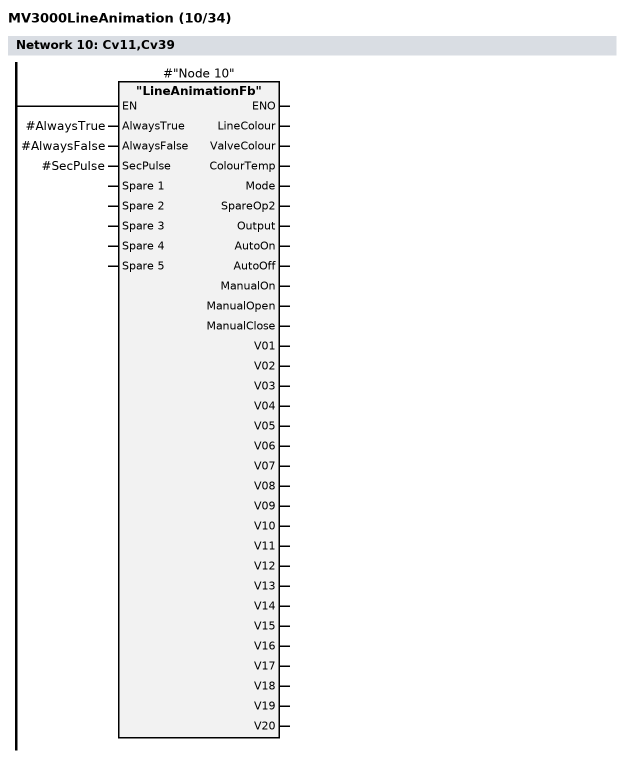
   RUNG wire#powerrail
      #"Node 10"(AlwaysTrue := #AlwaysTrue, AlwaysFalse := #AlwaysFalse, SecPulse := #SecPulse, "Spare 1" :=, "Spare 2" :=, "Spare 3" :=, "Spare 4" :=, "Spare 5" :=, LineColour =>, ValveColour =>, ColourTemp =>, Mode =>, SpareOp2 =>, Output =>, AutoOn =>, AutoOff =>, ManualOn =>, ManualOpen =>, ManualClose =>, V01 =>, V02 =>, V03 =>, V04 =>, V05 =>, V06 =>, V07 =>, V08 =>, V09 =>, V10 =>, V11 =>, V12 =>, V13 =>, V14 =>, V15 =>, V16 =>, V17 =>, V18 =>, V19 =>, V20 =>)
   END_RUNG
   // the same network as SCL:
   #"Node 10"(AlwaysTrue := #AlwaysTrue, AlwaysFalse := #AlwaysFalse, SecPulse := #SecPulse);   // "LineAnimationFb"
END_REGION

REGION Network 11: Cv12,Cv64, Cv26
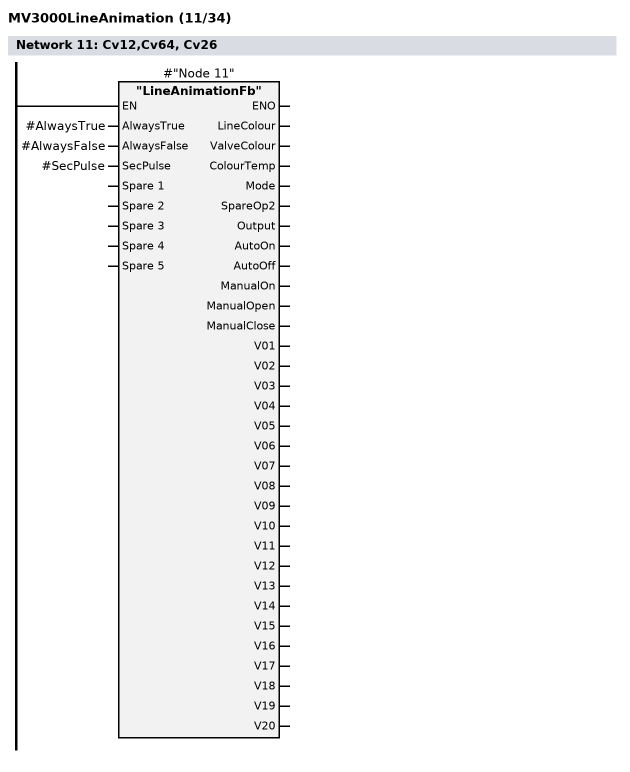
   RUNG wire#powerrail
      #"Node 11"(AlwaysTrue := #AlwaysTrue, AlwaysFalse := #AlwaysFalse, SecPulse := #SecPulse, "Spare 1" :=, "Spare 2" :=, "Spare 3" :=, "Spare 4" :=, "Spare 5" :=, LineColour =>, ValveColour =>, ColourTemp =>, Mode =>, SpareOp2 =>, Output =>, AutoOn =>, AutoOff =>, ManualOn =>, ManualOpen =>, ManualClose =>, V01 =>, V02 =>, V03 =>, V04 =>, V05 =>, V06 =>, V07 =>, V08 =>, V09 =>, V10 =>, V11 =>, V12 =>, V13 =>, V14 =>, V15 =>, V16 =>, V17 =>, V18 =>, V19 =>, V20 =>)
   END_RUNG
   // the same network as SCL:
   #"Node 11"(AlwaysTrue := #AlwaysTrue, AlwaysFalse := #AlwaysFalse, SecPulse := #SecPulse);   // "LineAnimationFb"
END_REGION

REGION Network 12: Cv31,Cv41
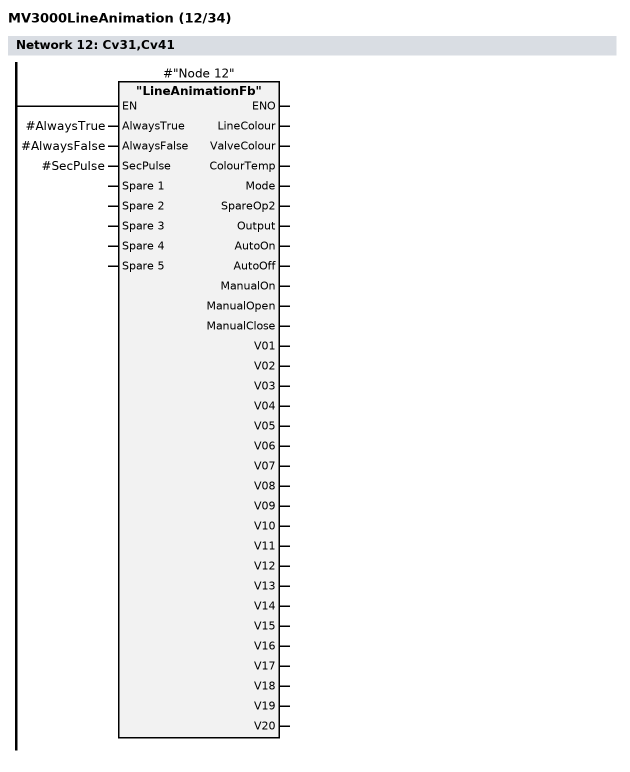
   RUNG wire#powerrail
      #"Node 12"(AlwaysTrue := #AlwaysTrue, AlwaysFalse := #AlwaysFalse, SecPulse := #SecPulse, "Spare 1" :=, "Spare 2" :=, "Spare 3" :=, "Spare 4" :=, "Spare 5" :=, LineColour =>, ValveColour =>, ColourTemp =>, Mode =>, SpareOp2 =>, Output =>, AutoOn =>, AutoOff =>, ManualOn =>, ManualOpen =>, ManualClose =>, V01 =>, V02 =>, V03 =>, V04 =>, V05 =>, V06 =>, V07 =>, V08 =>, V09 =>, V10 =>, V11 =>, V12 =>, V13 =>, V14 =>, V15 =>, V16 =>, V17 =>, V18 =>, V19 =>, V20 =>)
   END_RUNG
   // the same network as SCL:
   #"Node 12"(AlwaysTrue := #AlwaysTrue, AlwaysFalse := #AlwaysFalse, SecPulse := #SecPulse);   // "LineAnimationFb"
END_REGION

REGION Network 13: Fbov01, cV30 ,CV31 , CV 32 , CV33
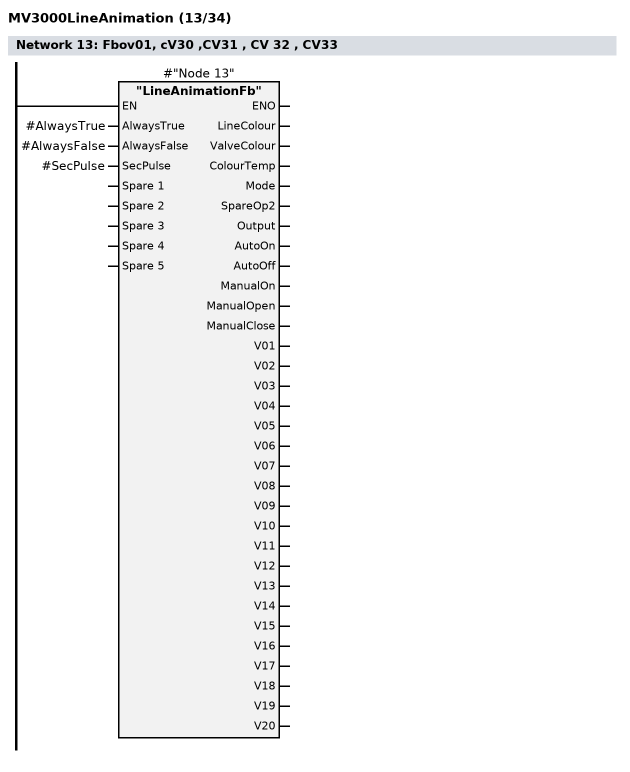
   RUNG wire#powerrail
      #"Node 13"(AlwaysTrue := #AlwaysTrue, AlwaysFalse := #AlwaysFalse, SecPulse := #SecPulse, "Spare 1" :=, "Spare 2" :=, "Spare 3" :=, "Spare 4" :=, "Spare 5" :=, LineColour =>, ValveColour =>, ColourTemp =>, Mode =>, SpareOp2 =>, Output =>, AutoOn =>, AutoOff =>, ManualOn =>, ManualOpen =>, ManualClose =>, V01 =>, V02 =>, V03 =>, V04 =>, V05 =>, V06 =>, V07 =>, V08 =>, V09 =>, V10 =>, V11 =>, V12 =>, V13 =>, V14 =>, V15 =>, V16 =>, V17 =>, V18 =>, V19 =>, V20 =>)
   END_RUNG
   // the same network as SCL:
   #"Node 13"(AlwaysTrue := #AlwaysTrue, AlwaysFalse := #AlwaysFalse, SecPulse := #SecPulse);   // "LineAnimationFb"
END_REGION

REGION Network 14: CV27 ,CV 28 ,CV 29
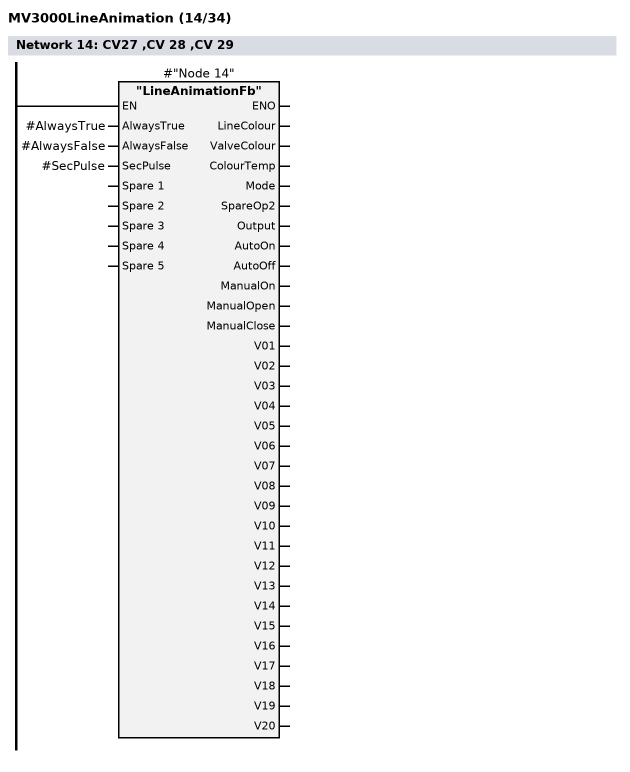
   RUNG wire#powerrail
      #"Node 14"(AlwaysTrue := #AlwaysTrue, AlwaysFalse := #AlwaysFalse, SecPulse := #SecPulse, "Spare 1" :=, "Spare 2" :=, "Spare 3" :=, "Spare 4" :=, "Spare 5" :=, LineColour =>, ValveColour =>, ColourTemp =>, Mode =>, SpareOp2 =>, Output =>, AutoOn =>, AutoOff =>, ManualOn =>, ManualOpen =>, ManualClose =>, V01 =>, V02 =>, V03 =>, V04 =>, V05 =>, V06 =>, V07 =>, V08 =>, V09 =>, V10 =>, V11 =>, V12 =>, V13 =>, V14 =>, V15 =>, V16 =>, V17 =>, V18 =>, V19 =>, V20 =>)
   END_RUNG
   // the same network as SCL:
   #"Node 14"(AlwaysTrue := #AlwaysTrue, AlwaysFalse := #AlwaysFalse, SecPulse := #SecPulse);   // "LineAnimationFb"
END_REGION

REGION Network 15: CV30 ,CV 33 ,CV 34,CV 35
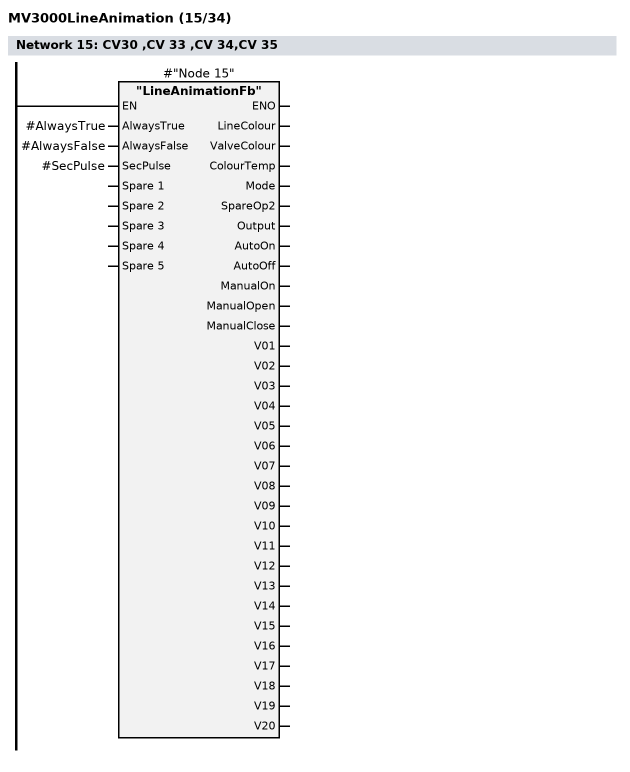
   RUNG wire#powerrail
      #"Node 15"(AlwaysTrue := #AlwaysTrue, AlwaysFalse := #AlwaysFalse, SecPulse := #SecPulse, "Spare 1" :=, "Spare 2" :=, "Spare 3" :=, "Spare 4" :=, "Spare 5" :=, LineColour =>, ValveColour =>, ColourTemp =>, Mode =>, SpareOp2 =>, Output =>, AutoOn =>, AutoOff =>, ManualOn =>, ManualOpen =>, ManualClose =>, V01 =>, V02 =>, V03 =>, V04 =>, V05 =>, V06 =>, V07 =>, V08 =>, V09 =>, V10 =>, V11 =>, V12 =>, V13 =>, V14 =>, V15 =>, V16 =>, V17 =>, V18 =>, V19 =>, V20 =>)
   END_RUNG
   // the same network as SCL:
   #"Node 15"(AlwaysTrue := #AlwaysTrue, AlwaysFalse := #AlwaysFalse, SecPulse := #SecPulse);   // "LineAnimationFb"
END_REGION

REGION Network 16: CV32 ,CV 36 ,CV 39,CV 40
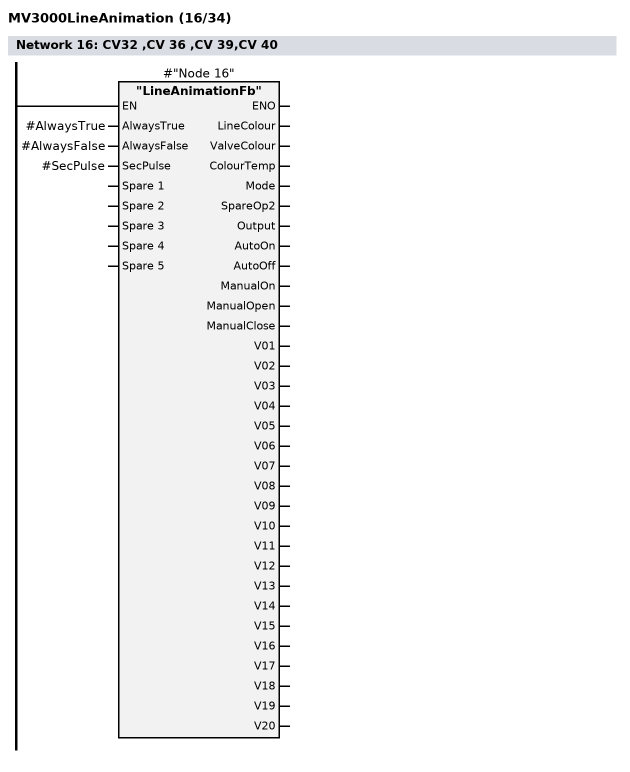
   RUNG wire#powerrail
      #"Node 16"(AlwaysTrue := #AlwaysTrue, AlwaysFalse := #AlwaysFalse, SecPulse := #SecPulse, "Spare 1" :=, "Spare 2" :=, "Spare 3" :=, "Spare 4" :=, "Spare 5" :=, LineColour =>, ValveColour =>, ColourTemp =>, Mode =>, SpareOp2 =>, Output =>, AutoOn =>, AutoOff =>, ManualOn =>, ManualOpen =>, ManualClose =>, V01 =>, V02 =>, V03 =>, V04 =>, V05 =>, V06 =>, V07 =>, V08 =>, V09 =>, V10 =>, V11 =>, V12 =>, V13 =>, V14 =>, V15 =>, V16 =>, V17 =>, V18 =>, V19 =>, V20 =>)
   END_RUNG
   // the same network as SCL:
   #"Node 16"(AlwaysTrue := #AlwaysTrue, AlwaysFalse := #AlwaysFalse, SecPulse := #SecPulse);   // "LineAnimationFb"
END_REGION

REGION Network 17: CV40 ,CV41 ,CV 42 ,CV 43,CV 44
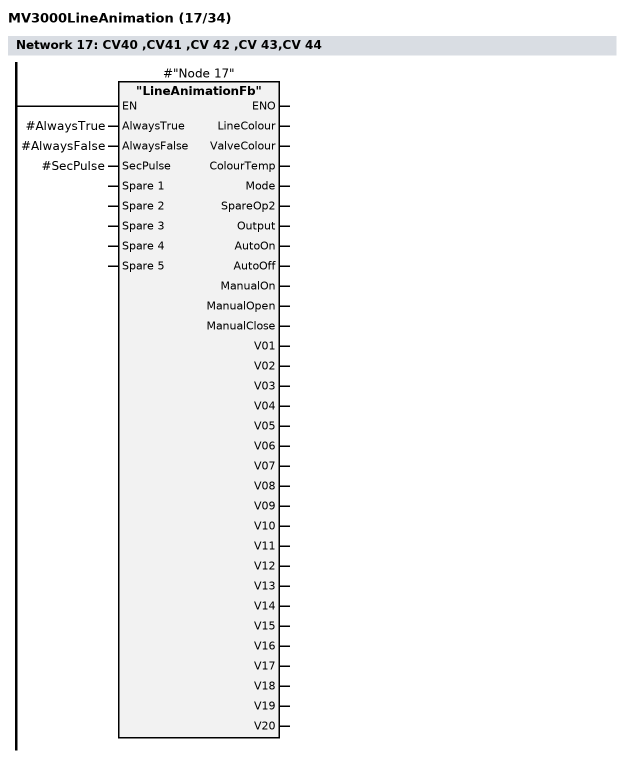
   RUNG wire#powerrail
      #"Node 17"(AlwaysTrue := #AlwaysTrue, AlwaysFalse := #AlwaysFalse, SecPulse := #SecPulse, "Spare 1" :=, "Spare 2" :=, "Spare 3" :=, "Spare 4" :=, "Spare 5" :=, LineColour =>, ValveColour =>, ColourTemp =>, Mode =>, SpareOp2 =>, Output =>, AutoOn =>, AutoOff =>, ManualOn =>, ManualOpen =>, ManualClose =>, V01 =>, V02 =>, V03 =>, V04 =>, V05 =>, V06 =>, V07 =>, V08 =>, V09 =>, V10 =>, V11 =>, V12 =>, V13 =>, V14 =>, V15 =>, V16 =>, V17 =>, V18 =>, V19 =>, V20 =>)
   END_RUNG
   // the same network as SCL:
   #"Node 17"(AlwaysTrue := #AlwaysTrue, AlwaysFalse := #AlwaysFalse, SecPulse := #SecPulse);   // "LineAnimationFb"
END_REGION

REGION Network 18: CV43 ,CV47 ,CV 48 ,CV 49,CV 50
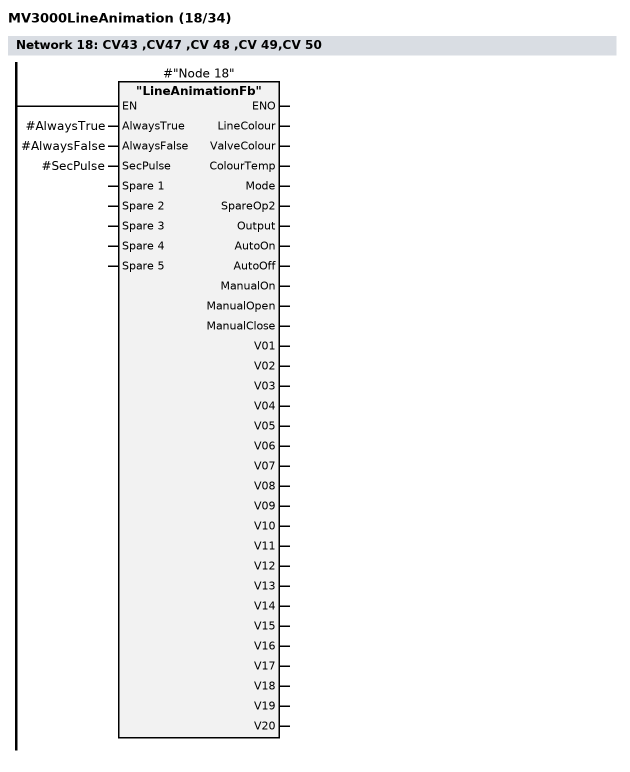
   RUNG wire#powerrail
      #"Node 18"(AlwaysTrue := #AlwaysTrue, AlwaysFalse := #AlwaysFalse, SecPulse := #SecPulse, "Spare 1" :=, "Spare 2" :=, "Spare 3" :=, "Spare 4" :=, "Spare 5" :=, LineColour =>, ValveColour =>, ColourTemp =>, Mode =>, SpareOp2 =>, Output =>, AutoOn =>, AutoOff =>, ManualOn =>, ManualOpen =>, ManualClose =>, V01 =>, V02 =>, V03 =>, V04 =>, V05 =>, V06 =>, V07 =>, V08 =>, V09 =>, V10 =>, V11 =>, V12 =>, V13 =>, V14 =>, V15 =>, V16 =>, V17 =>, V18 =>, V19 =>, V20 =>)
   END_RUNG
   // the same network as SCL:
   #"Node 18"(AlwaysTrue := #AlwaysTrue, AlwaysFalse := #AlwaysFalse, SecPulse := #SecPulse);   // "LineAnimationFb"
END_REGION

REGION Network 19: CV49 ,CV53 ,CV 54 ,CV 55,CV 56
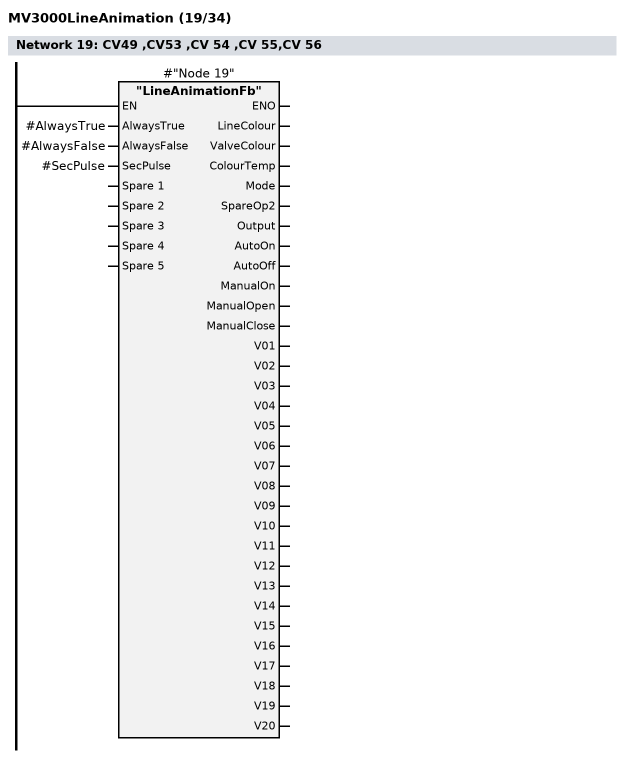
   RUNG wire#powerrail
      #"Node 19"(AlwaysTrue := #AlwaysTrue, AlwaysFalse := #AlwaysFalse, SecPulse := #SecPulse, "Spare 1" :=, "Spare 2" :=, "Spare 3" :=, "Spare 4" :=, "Spare 5" :=, LineColour =>, ValveColour =>, ColourTemp =>, Mode =>, SpareOp2 =>, Output =>, AutoOn =>, AutoOff =>, ManualOn =>, ManualOpen =>, ManualClose =>, V01 =>, V02 =>, V03 =>, V04 =>, V05 =>, V06 =>, V07 =>, V08 =>, V09 =>, V10 =>, V11 =>, V12 =>, V13 =>, V14 =>, V15 =>, V16 =>, V17 =>, V18 =>, V19 =>, V20 =>)
   END_RUNG
   // the same network as SCL:
   #"Node 19"(AlwaysTrue := #AlwaysTrue, AlwaysFalse := #AlwaysFalse, SecPulse := #SecPulse);   // "LineAnimationFb"
END_REGION

REGION Network 20: Cv55,Cv61, Cv62
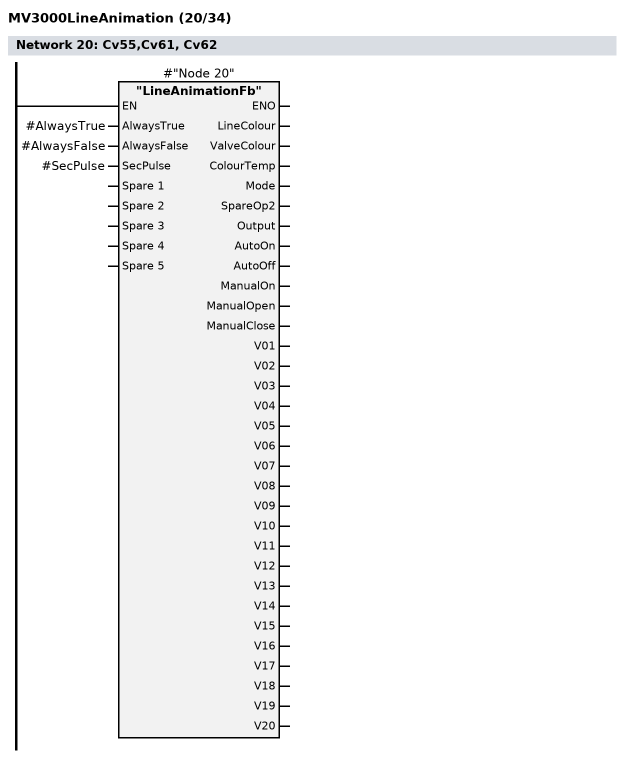
   RUNG wire#powerrail
      #"Node 20"(AlwaysTrue := #AlwaysTrue, AlwaysFalse := #AlwaysFalse, SecPulse := #SecPulse, "Spare 1" :=, "Spare 2" :=, "Spare 3" :=, "Spare 4" :=, "Spare 5" :=, LineColour =>, ValveColour =>, ColourTemp =>, Mode =>, SpareOp2 =>, Output =>, AutoOn =>, AutoOff =>, ManualOn =>, ManualOpen =>, ManualClose =>, V01 =>, V02 =>, V03 =>, V04 =>, V05 =>, V06 =>, V07 =>, V08 =>, V09 =>, V10 =>, V11 =>, V12 =>, V13 =>, V14 =>, V15 =>, V16 =>, V17 =>, V18 =>, V19 =>, V20 =>)
   END_RUNG
   // the same network as SCL:
   #"Node 20"(AlwaysTrue := #AlwaysTrue, AlwaysFalse := #AlwaysFalse, SecPulse := #SecPulse);   // "LineAnimationFb"
END_REGION

REGION Network 21: Cv59,Cv60, Cv61
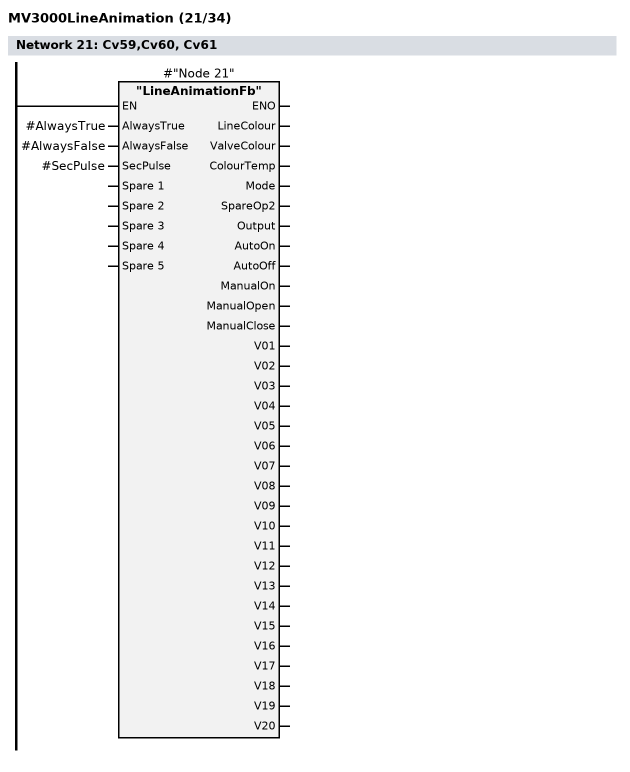
   RUNG wire#powerrail
      #"Node 21"(AlwaysTrue := #AlwaysTrue, AlwaysFalse := #AlwaysFalse, SecPulse := #SecPulse, "Spare 1" :=, "Spare 2" :=, "Spare 3" :=, "Spare 4" :=, "Spare 5" :=, LineColour =>, ValveColour =>, ColourTemp =>, Mode =>, SpareOp2 =>, Output =>, AutoOn =>, AutoOff =>, ManualOn =>, ManualOpen =>, ManualClose =>, V01 =>, V02 =>, V03 =>, V04 =>, V05 =>, V06 =>, V07 =>, V08 =>, V09 =>, V10 =>, V11 =>, V12 =>, V13 =>, V14 =>, V15 =>, V16 =>, V17 =>, V18 =>, V19 =>, V20 =>)
   END_RUNG
   // the same network as SCL:
   #"Node 21"(AlwaysTrue := #AlwaysTrue, AlwaysFalse := #AlwaysFalse, SecPulse := #SecPulse);   // "LineAnimationFb"
END_REGION

REGION Network 22: Cv56,Cv58, Cv57
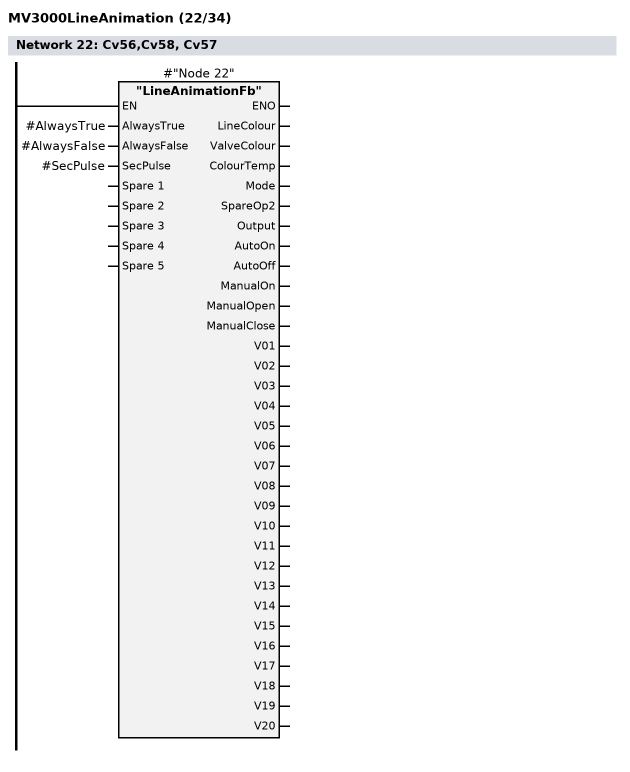
   RUNG wire#powerrail
      #"Node 22"(AlwaysTrue := #AlwaysTrue, AlwaysFalse := #AlwaysFalse, SecPulse := #SecPulse, "Spare 1" :=, "Spare 2" :=, "Spare 3" :=, "Spare 4" :=, "Spare 5" :=, LineColour =>, ValveColour =>, ColourTemp =>, Mode =>, SpareOp2 =>, Output =>, AutoOn =>, AutoOff =>, ManualOn =>, ManualOpen =>, ManualClose =>, V01 =>, V02 =>, V03 =>, V04 =>, V05 =>, V06 =>, V07 =>, V08 =>, V09 =>, V10 =>, V11 =>, V12 =>, V13 =>, V14 =>, V15 =>, V16 =>, V17 =>, V18 =>, V19 =>, V20 =>)
   END_RUNG
   // the same network as SCL:
   #"Node 22"(AlwaysTrue := #AlwaysTrue, AlwaysFalse := #AlwaysFalse, SecPulse := #SecPulse);   // "LineAnimationFb"
END_REGION

REGION Network 23: Cv50,Cv51, Cv52,Cv53
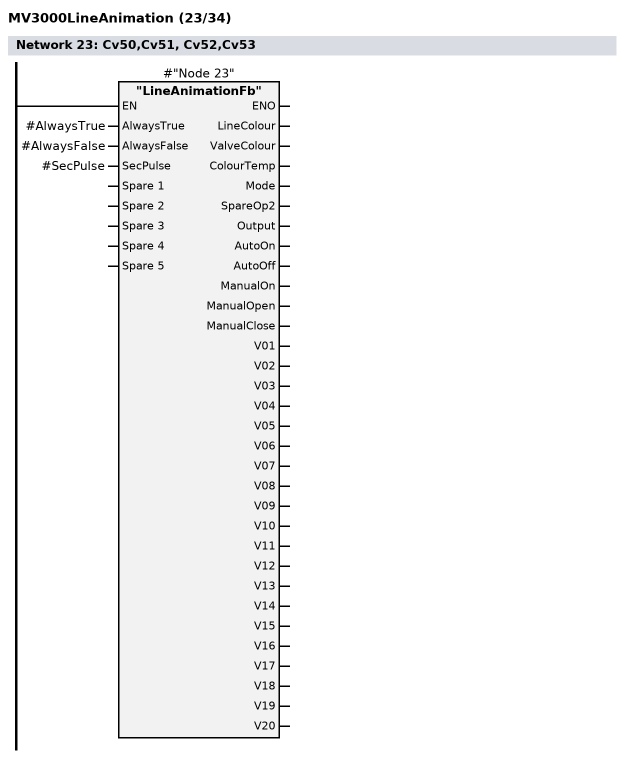
   RUNG wire#powerrail
      #"Node 23"(AlwaysTrue := #AlwaysTrue, AlwaysFalse := #AlwaysFalse, SecPulse := #SecPulse, "Spare 1" :=, "Spare 2" :=, "Spare 3" :=, "Spare 4" :=, "Spare 5" :=, LineColour =>, ValveColour =>, ColourTemp =>, Mode =>, SpareOp2 =>, Output =>, AutoOn =>, AutoOff =>, ManualOn =>, ManualOpen =>, ManualClose =>, V01 =>, V02 =>, V03 =>, V04 =>, V05 =>, V06 =>, V07 =>, V08 =>, V09 =>, V10 =>, V11 =>, V12 =>, V13 =>, V14 =>, V15 =>, V16 =>, V17 =>, V18 =>, V19 =>, V20 =>)
   END_RUNG
   // the same network as SCL:
   #"Node 23"(AlwaysTrue := #AlwaysTrue, AlwaysFalse := #AlwaysFalse, SecPulse := #SecPulse);   // "LineAnimationFb"
END_REGION

REGION Network 24: Cv44,Cv45, Cv46,Cv47
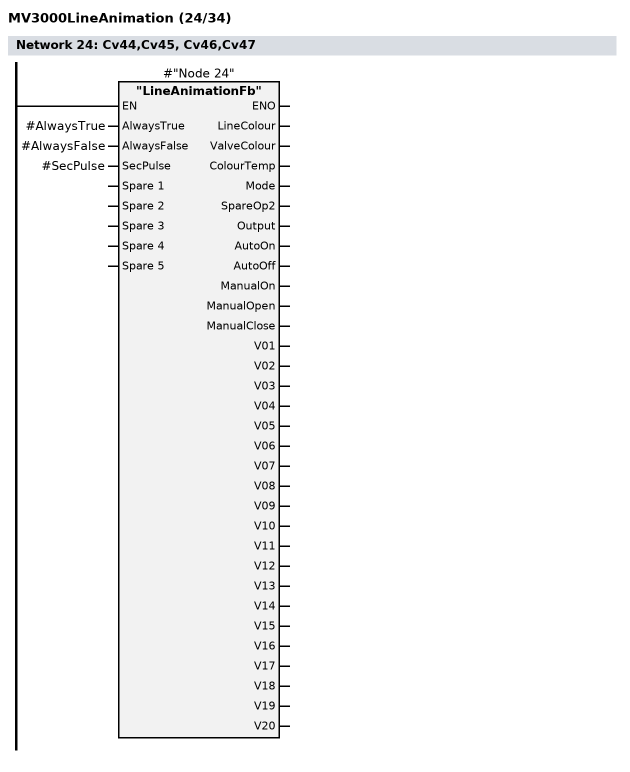
   RUNG wire#powerrail
      #"Node 24"(AlwaysTrue := #AlwaysTrue, AlwaysFalse := #AlwaysFalse, SecPulse := #SecPulse, "Spare 1" :=, "Spare 2" :=, "Spare 3" :=, "Spare 4" :=, "Spare 5" :=, LineColour =>, ValveColour =>, ColourTemp =>, Mode =>, SpareOp2 =>, Output =>, AutoOn =>, AutoOff =>, ManualOn =>, ManualOpen =>, ManualClose =>, V01 =>, V02 =>, V03 =>, V04 =>, V05 =>, V06 =>, V07 =>, V08 =>, V09 =>, V10 =>, V11 =>, V12 =>, V13 =>, V14 =>, V15 =>, V16 =>, V17 =>, V18 =>, V19 =>, V20 =>)
   END_RUNG
   // the same network as SCL:
   #"Node 24"(AlwaysTrue := #AlwaysTrue, AlwaysFalse := #AlwaysFalse, SecPulse := #SecPulse);   // "LineAnimationFb"
END_REGION

REGION Network 25: Cv36,Cv37, Cv38
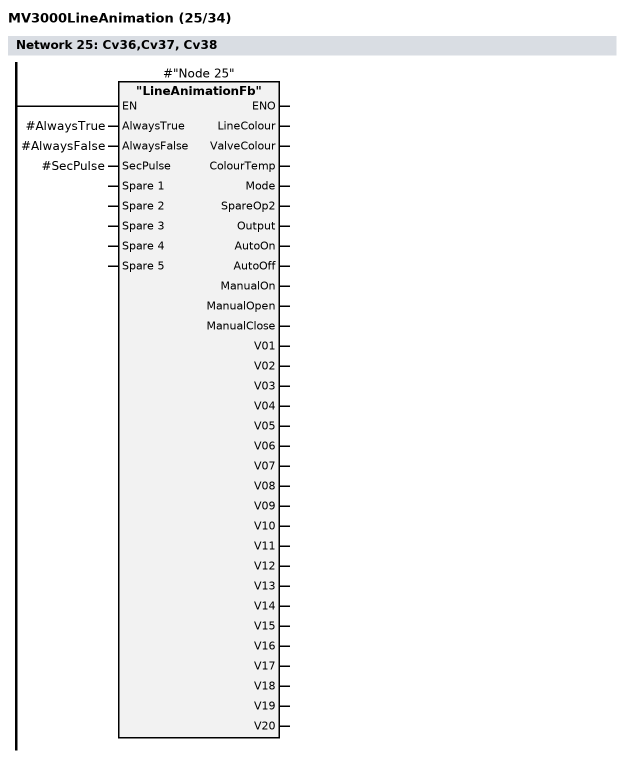
   RUNG wire#powerrail
      #"Node 25"(AlwaysTrue := #AlwaysTrue, AlwaysFalse := #AlwaysFalse, SecPulse := #SecPulse, "Spare 1" :=, "Spare 2" :=, "Spare 3" :=, "Spare 4" :=, "Spare 5" :=, LineColour =>, ValveColour =>, ColourTemp =>, Mode =>, SpareOp2 =>, Output =>, AutoOn =>, AutoOff =>, ManualOn =>, ManualOpen =>, ManualClose =>, V01 =>, V02 =>, V03 =>, V04 =>, V05 =>, V06 =>, V07 =>, V08 =>, V09 =>, V10 =>, V11 =>, V12 =>, V13 =>, V14 =>, V15 =>, V16 =>, V17 =>, V18 =>, V19 =>, V20 =>)
   END_RUNG
   // the same network as SCL:
   #"Node 25"(AlwaysTrue := #AlwaysTrue, AlwaysFalse := #AlwaysFalse, SecPulse := #SecPulse);   // "LineAnimationFb"
END_REGION

REGION Network 26: Cv30,Cv33, Cv34,Cv35
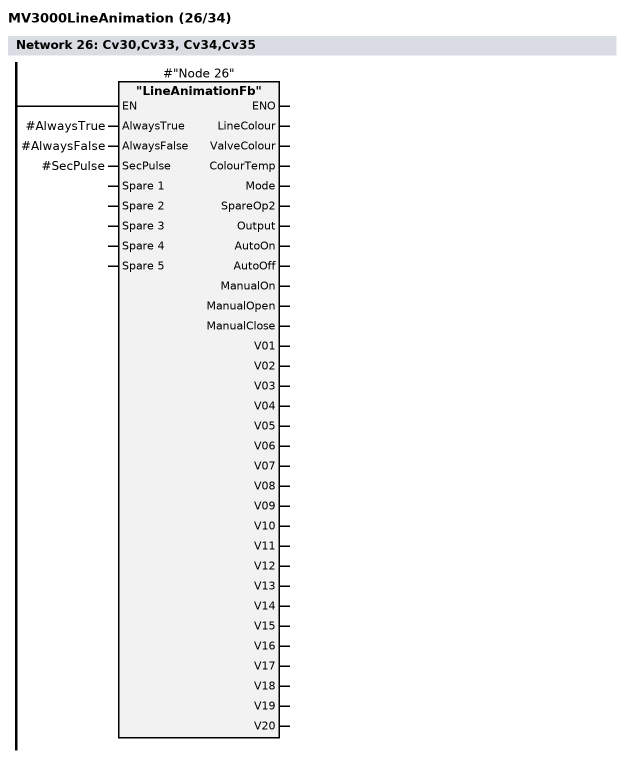
   RUNG wire#powerrail
      #"Node 26"(AlwaysTrue := #AlwaysTrue, AlwaysFalse := #AlwaysFalse, SecPulse := #SecPulse, "Spare 1" :=, "Spare 2" :=, "Spare 3" :=, "Spare 4" :=, "Spare 5" :=, LineColour =>, ValveColour =>, ColourTemp =>, Mode =>, SpareOp2 =>, Output =>, AutoOn =>, AutoOff =>, ManualOn =>, ManualOpen =>, ManualClose =>, V01 =>, V02 =>, V03 =>, V04 =>, V05 =>, V06 =>, V07 =>, V08 =>, V09 =>, V10 =>, V11 =>, V12 =>, V13 =>, V14 =>, V15 =>, V16 =>, V17 =>, V18 =>, V19 =>, V20 =>)
   END_RUNG
   // the same network as SCL:
   #"Node 26"(AlwaysTrue := #AlwaysTrue, AlwaysFalse := #AlwaysFalse, SecPulse := #SecPulse);   // "LineAnimationFb"
END_REGION

REGION Network 27: Cv28, Cv34,Cv37,Cv45,Cv51, Cv57,Cv60
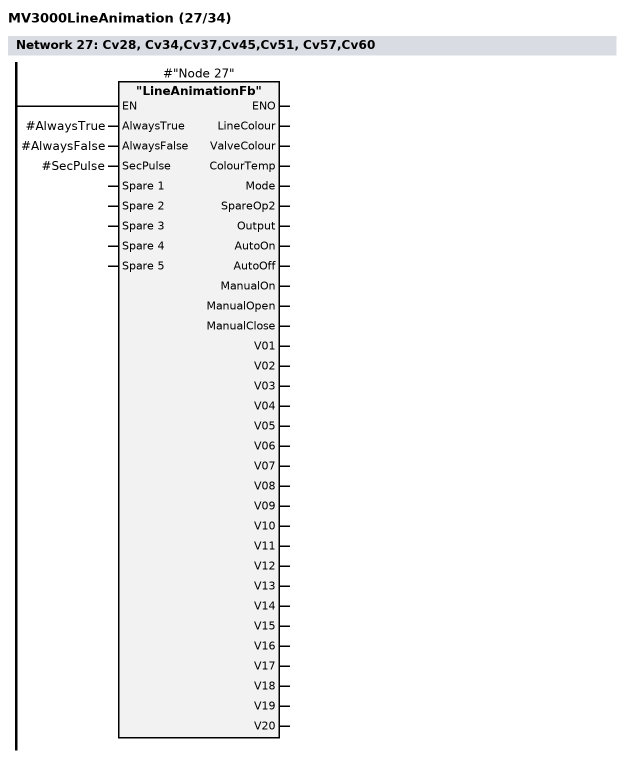
   RUNG wire#powerrail
      #"Node 27"(AlwaysTrue := #AlwaysTrue, AlwaysFalse := #AlwaysFalse, SecPulse := #SecPulse, "Spare 1" :=, "Spare 2" :=, "Spare 3" :=, "Spare 4" :=, "Spare 5" :=, LineColour =>, ValveColour =>, ColourTemp =>, Mode =>, SpareOp2 =>, Output =>, AutoOn =>, AutoOff =>, ManualOn =>, ManualOpen =>, ManualClose =>, V01 =>, V02 =>, V03 =>, V04 =>, V05 =>, V06 =>, V07 =>, V08 =>, V09 =>, V10 =>, V11 =>, V12 =>, V13 =>, V14 =>, V15 =>, V16 =>, V17 =>, V18 =>, V19 =>, V20 =>)
   END_RUNG
   // the same network as SCL:
   #"Node 27"(AlwaysTrue := #AlwaysTrue, AlwaysFalse := #AlwaysFalse, SecPulse := #SecPulse);   // "LineAnimationFb"
END_REGION

REGION Network 28: Cv22, Cv25,Cv19,Cv20,Cv29,Cv35, Cv38,C46 ,Cv52 ,Cv58 ,Cv59
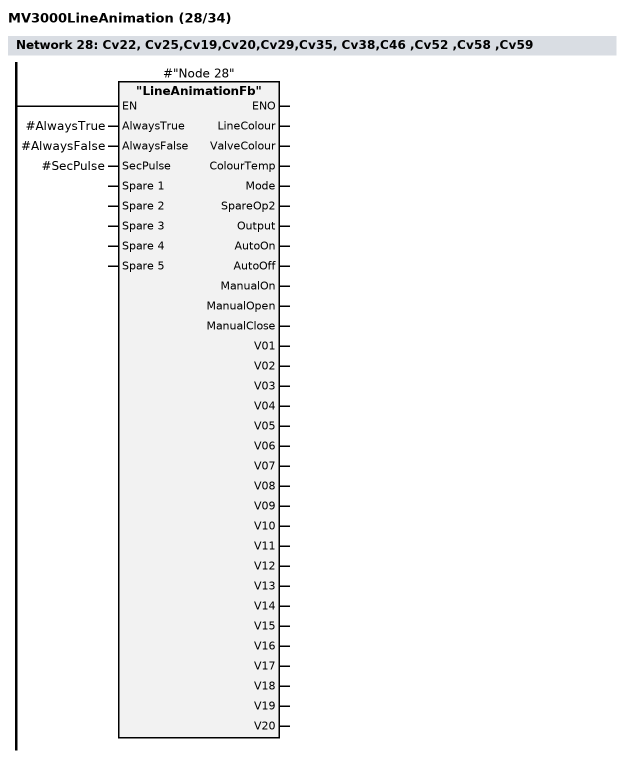
   RUNG wire#powerrail
      #"Node 28"(AlwaysTrue := #AlwaysTrue, AlwaysFalse := #AlwaysFalse, SecPulse := #SecPulse, "Spare 1" :=, "Spare 2" :=, "Spare 3" :=, "Spare 4" :=, "Spare 5" :=, LineColour =>, ValveColour =>, ColourTemp =>, Mode =>, SpareOp2 =>, Output =>, AutoOn =>, AutoOff =>, ManualOn =>, ManualOpen =>, ManualClose =>, V01 =>, V02 =>, V03 =>, V04 =>, V05 =>, V06 =>, V07 =>, V08 =>, V09 =>, V10 =>, V11 =>, V12 =>, V13 =>, V14 =>, V15 =>, V16 =>, V17 =>, V18 =>, V19 =>, V20 =>)
   END_RUNG
   // the same network as SCL:
   #"Node 28"(AlwaysTrue := #AlwaysTrue, AlwaysFalse := #AlwaysFalse, SecPulse := #SecPulse);   // "LineAnimationFb"
END_REGION

REGION Network 29: Cv01,Cv04
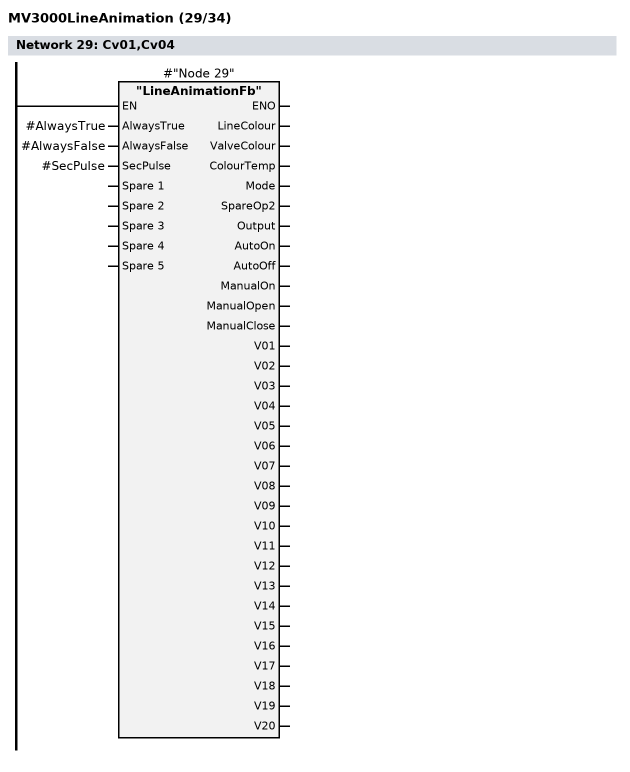
   RUNG wire#powerrail
      #"Node 29"(AlwaysTrue := #AlwaysTrue, AlwaysFalse := #AlwaysFalse, SecPulse := #SecPulse, "Spare 1" :=, "Spare 2" :=, "Spare 3" :=, "Spare 4" :=, "Spare 5" :=, LineColour =>, ValveColour =>, ColourTemp =>, Mode =>, SpareOp2 =>, Output =>, AutoOn =>, AutoOff =>, ManualOn =>, ManualOpen =>, ManualClose =>, V01 =>, V02 =>, V03 =>, V04 =>, V05 =>, V06 =>, V07 =>, V08 =>, V09 =>, V10 =>, V11 =>, V12 =>, V13 =>, V14 =>, V15 =>, V16 =>, V17 =>, V18 =>, V19 =>, V20 =>)
   END_RUNG
   // the same network as SCL:
   #"Node 29"(AlwaysTrue := #AlwaysTrue, AlwaysFalse := #AlwaysFalse, SecPulse := #SecPulse);   // "LineAnimationFb"
END_REGION

REGION Network 30: Cv06,Cv09
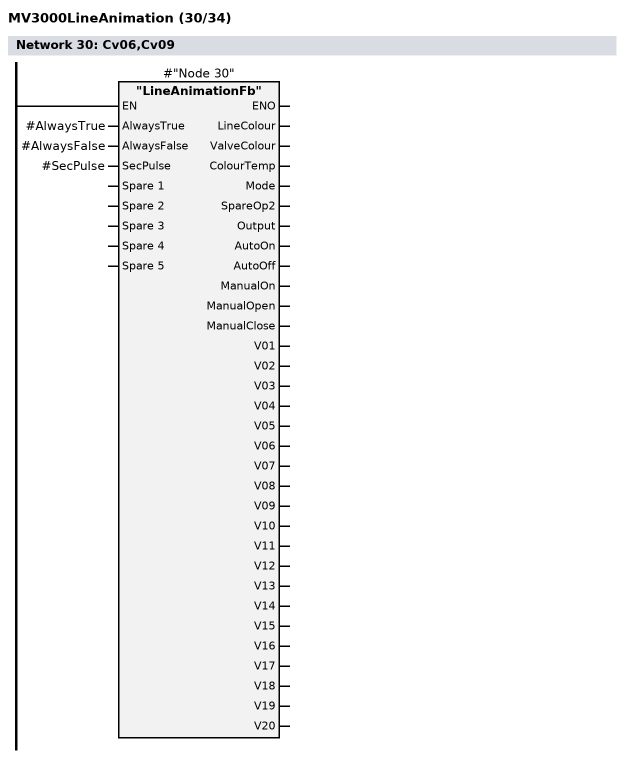
   RUNG wire#powerrail
      #"Node 30"(AlwaysTrue := #AlwaysTrue, AlwaysFalse := #AlwaysFalse, SecPulse := #SecPulse, "Spare 1" :=, "Spare 2" :=, "Spare 3" :=, "Spare 4" :=, "Spare 5" :=, LineColour =>, ValveColour =>, ColourTemp =>, Mode =>, SpareOp2 =>, Output =>, AutoOn =>, AutoOff =>, ManualOn =>, ManualOpen =>, ManualClose =>, V01 =>, V02 =>, V03 =>, V04 =>, V05 =>, V06 =>, V07 =>, V08 =>, V09 =>, V10 =>, V11 =>, V12 =>, V13 =>, V14 =>, V15 =>, V16 =>, V17 =>, V18 =>, V19 =>, V20 =>)
   END_RUNG
   // the same network as SCL:
   #"Node 30"(AlwaysTrue := #AlwaysTrue, AlwaysFalse := #AlwaysFalse, SecPulse := #SecPulse);   // "LineAnimationFb"
END_REGION

REGION Network 31: Cv06,Cv09 ,Cv08
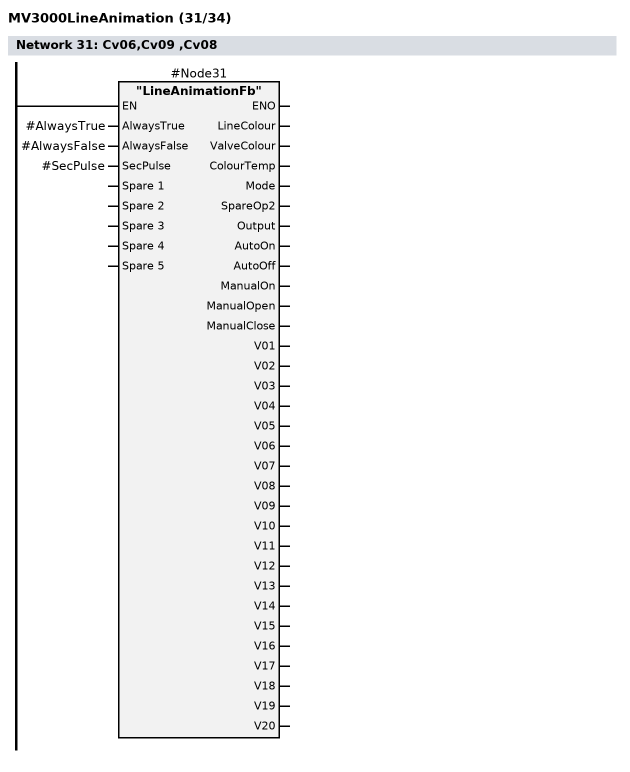
   RUNG wire#powerrail
      #Node31(AlwaysTrue := #AlwaysTrue, AlwaysFalse := #AlwaysFalse, SecPulse := #SecPulse, "Spare 1" :=, "Spare 2" :=, "Spare 3" :=, "Spare 4" :=, "Spare 5" :=, LineColour =>, ValveColour =>, ColourTemp =>, Mode =>, SpareOp2 =>, Output =>, AutoOn =>, AutoOff =>, ManualOn =>, ManualOpen =>, ManualClose =>, V01 =>, V02 =>, V03 =>, V04 =>, V05 =>, V06 =>, V07 =>, V08 =>, V09 =>, V10 =>, V11 =>, V12 =>, V13 =>, V14 =>, V15 =>, V16 =>, V17 =>, V18 =>, V19 =>, V20 =>)
   END_RUNG
   // the same network as SCL:
   #Node31(AlwaysTrue := #AlwaysTrue, AlwaysFalse := #AlwaysFalse, SecPulse := #SecPulse);   // "LineAnimationFb"
END_REGION

REGION Network 32: Cv05,Cv24
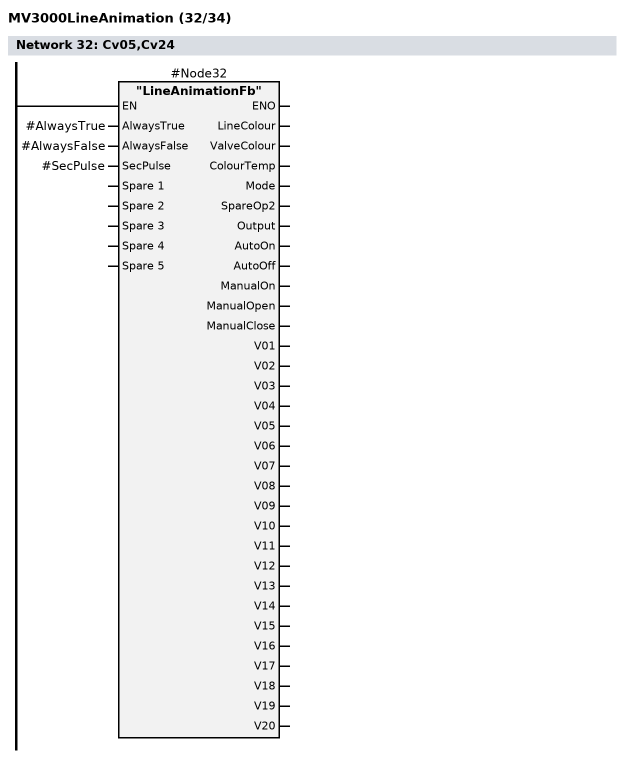
   RUNG wire#powerrail
      #Node32(AlwaysTrue := #AlwaysTrue, AlwaysFalse := #AlwaysFalse, SecPulse := #SecPulse, "Spare 1" :=, "Spare 2" :=, "Spare 3" :=, "Spare 4" :=, "Spare 5" :=, LineColour =>, ValveColour =>, ColourTemp =>, Mode =>, SpareOp2 =>, Output =>, AutoOn =>, AutoOff =>, ManualOn =>, ManualOpen =>, ManualClose =>, V01 =>, V02 =>, V03 =>, V04 =>, V05 =>, V06 =>, V07 =>, V08 =>, V09 =>, V10 =>, V11 =>, V12 =>, V13 =>, V14 =>, V15 =>, V16 =>, V17 =>, V18 =>, V19 =>, V20 =>)
   END_RUNG
   // the same network as SCL:
   #Node32(AlwaysTrue := #AlwaysTrue, AlwaysFalse := #AlwaysFalse, SecPulse := #SecPulse);   // "LineAnimationFb"
END_REGION

REGION Network 33: CvFbv01,Cv26
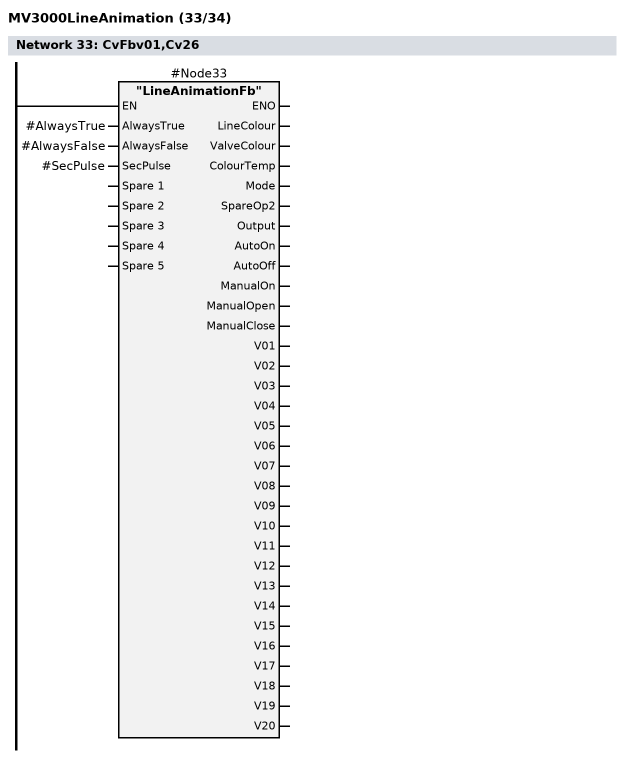
   RUNG wire#powerrail
      #Node33(AlwaysTrue := #AlwaysTrue, AlwaysFalse := #AlwaysFalse, SecPulse := #SecPulse, "Spare 1" :=, "Spare 2" :=, "Spare 3" :=, "Spare 4" :=, "Spare 5" :=, LineColour =>, ValveColour =>, ColourTemp =>, Mode =>, SpareOp2 =>, Output =>, AutoOn =>, AutoOff =>, ManualOn =>, ManualOpen =>, ManualClose =>, V01 =>, V02 =>, V03 =>, V04 =>, V05 =>, V06 =>, V07 =>, V08 =>, V09 =>, V10 =>, V11 =>, V12 =>, V13 =>, V14 =>, V15 =>, V16 =>, V17 =>, V18 =>, V19 =>, V20 =>)
   END_RUNG
   // the same network as SCL:
   #Node33(AlwaysTrue := #AlwaysTrue, AlwaysFalse := #AlwaysFalse, SecPulse := #SecPulse);   // "LineAnimationFb"
END_REGION

REGION Network 34: Cv42,Cv54,Cv48
